Staubli VAL3: uniqueStr.pgx

public program uniqueStr(string& x_sInput[], string& x_sResult[])
  local num l_nCoutner
  local num l_nElement
  local num l_nLength
  local string l_sString
  local num l_nBuffer
  local bool l_bDone
  local bool l_bFound
  local num l_nMarker
begin

  l_nLength = size(x_sInput)
  l_nCoutner = 0
  resize(x_sResult,1,1)

  for l_nElement = 0 to l_nLength-1
    l_bFound = false
    if l_nElement == 0
      append(x_sResult)
      x_sResult[size(x_sResult)-1] = x_sInput[l_nElement]
    else

      for l_nBuffer = 0 to size(x_sResult)-1
        if x_sInput[l_nElement] != x_sResult[l_nBuffer]
          l_bFound = false
        else
          // break out of for-loop
          l_bFound = true
          l_nBuffer = size(x_sResult)+1
          l_nMarker = l_nBuffer
        endIf

      endFor

      if l_bFound == false
        append(x_sResult)
        x_sResult[size(x_sResult)-1] = x_sInput[l_nElement]
      endIf

   endIf

  endFor

  delete(x_sResult[0])

end
